% RSLogix 500 project Lab 2 code int.RSS, saved by version 8.30.00.16 %
PROJECT "UNTITLED"    % processor: Bul.1763 MicroLogix 1100 Series B %

PROGRAM FILES
  LAD 2   10 rungs

DATA FILES
  O0 OUTPUT  4 elements
  I1 INPUT  6 elements
  S2 STATUS  66 elements
  B3 BINARY  1 elements
  T4 TIMER  1 elements
  C5 COUNTER  1 elements
  R6 CONTROL  1 elements
  N7 INTEGER  1 elements
  F8 FLOAT  1 elements

LADDER 2
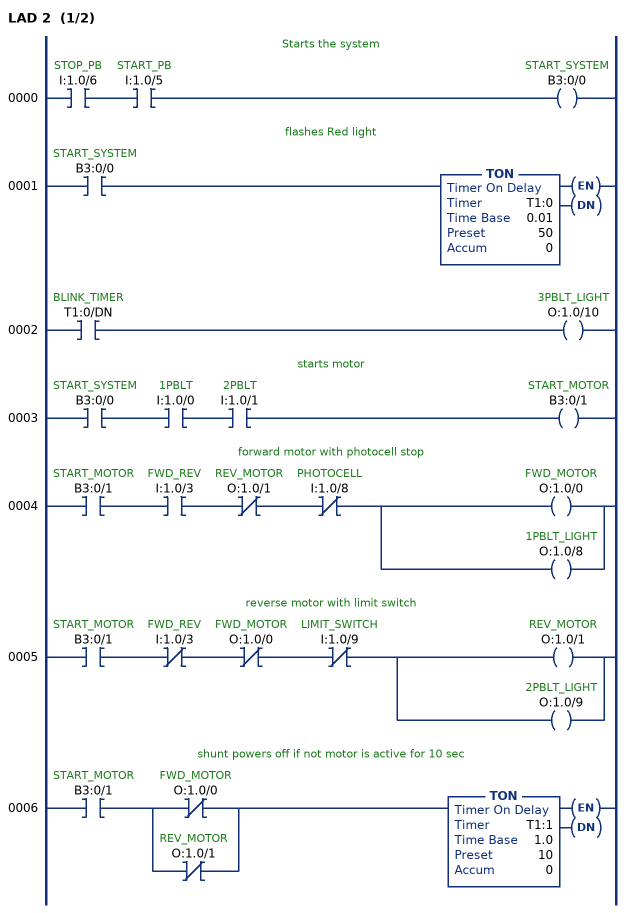
% Rung: 0 %  % edit flag set %
% Starts the system %
SOR XIC I:1.0/6 XIC I:1.0/5 OTE B3:0/0 EOR
%   I:1.0/6  STOP_PB %
%   I:1.0/5  START_PB %
%   B3:0/0  START_SYSTEM %
% Rung: 1 %  % edit flag set %
% flashes Red light %
SOR XIC B3:0/0 TON T1:0 0.01 50 0 EOR
%   B3:0/0  START_SYSTEM %
% Rung: 2 %  % edit flag set %
SOR XIC T1:0/DN OTE O:1.0/10 EOR
%   T1:0/DN  BLINK_TIMER %
%   O:1.0/10  3PBLT_LIGHT %
% Rung: 3 %  % edit flag set %
% starts motor %
SOR XIC B3:0/0 XIC I:1.0/0 XIC I:1.0/1 OTE B3:0/1 EOR
%   B3:0/0  START_SYSTEM %
%   I:1.0/0  1PBLT %
%   I:1.0/1  2PBLT %
%   B3:0/1  START_MOTOR %
% Rung: 4 %  % edit flag set %
% forward motor with photocell stop %
SOR XIC B3:0/1 XIC I:1.0/3 XIO O:1.0/1 XIO I:1.0/8 BST OTE O:1.0/0 NXB OTE O:1.0/8 BND EOR
%   B3:0/1  START_MOTOR %
%   I:1.0/3  FWD_REV %
%   O:1.0/1  REV_MOTOR %
%   I:1.0/8  PHOTOCELL %
%   O:1.0/0  FWD_MOTOR %
%   O:1.0/8  1PBLT_LIGHT %
% Rung: 5 %  % edit flag set %
% reverse motor with limit switch %
SOR XIC B3:0/1 XIO I:1.0/3 XIO O:1.0/0 XIO I:1.0/9 BST OTE O:1.0/1 NXB OTE O:1.0/9 BND EOR
%   B3:0/1  START_MOTOR %
%   I:1.0/3  FWD_REV %
%   O:1.0/0  FWD_MOTOR %
%   I:1.0/9  LIMIT_SWITCH %
%   O:1.0/1  REV_MOTOR %
%   O:1.0/9  2PBLT_LIGHT %
% Rung: 6 %  % edit flag set %
% shunt powers off if not motor is active for 10 sec %
SOR XIC B3:0/1 BST XIO O:1.0/0 NXB XIO O:1.0/1 BND TON T1:1 1.0 10 0 EOR
%   B3:0/1  START_MOTOR %
%   O:1.0/0  FWD_MOTOR %
%   O:1.0/1  REV_MOTOR %

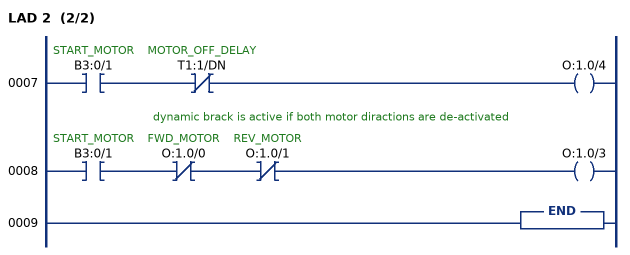
% Rung: 7 %  % edit flag set %
SOR XIC B3:0/1 XIO T1:1/DN OTE O:1.0/4 EOR
%   B3:0/1  START_MOTOR %
%   T1:1/DN  MOTOR_OFF_DELAY %
% Rung: 8 %  % edit flag set %
% dynamic brack is active if both motor diractions are de-activated %
SOR XIC B3:0/1 XIO O:1.0/0 XIO O:1.0/1 OTE O:1.0/3 EOR
%   B3:0/1  START_MOTOR %
%   O:1.0/0  FWD_MOTOR %
%   O:1.0/1  REV_MOTOR %
% Rung: 9 %
SOR END EOR
